Staubli VAL3: Delete.pgx

program Delete()
  local string l_sYesNo[2]
  local num l_i
begin
  //删除
  l_sYesNo[0]="是"
  l_sYesNo[1]="否"
  switch nPage
    case 0
      call user:questionDialog("是否删除此路径?",l_sYesNo,l_i)
      if l_i==0 or l_i==1
        if sFileList[nSelected]!=""
          libDelete(sFolder+sFileList[nSelected])
          delete(sFileList[nSelected])
          bListRefresh=true
        endIf
      endIf
    break
    case 1
      call user:questionDialog("是否删除此点?",l_sYesNo,l_i)
      if l_i==0 or l_i==1
        if sFileList[nSelected]!=""
          delete(prd:pDemo[nSelected])
          delete(prd:sPtParameter[nSelected])
          bListRefresh=true
        endIf
      endIf
    break
  endSwitch

  bUserRefresh=true
end
